// TIA Portal V21 export
DATA_BLOCK "Trend"   // DB5
{ S7_Optimized_Access := 'TRUE' }
// stored: MemoryReserve 100
   VAR
      T : Array[0.."K_NumTrends"] of "Std_Trend";
   END_VAR
BEGIN
   T[0].Valore1 := 0.0;
   T[0].Valore2 := 0.0;
   T[0].Valore3 := 0.0;
   T[0].Valore4 := 0.0;
   T[0].Valore5 := 0.0;
   T[0].Valore6 := 0.0;
   T[0].Valore7 := 0.0;
   T[0].Valore8 := 0.0;
   T[0].AsseY_SinistroMin := 0;
   T[0].AsseY_SinistroMax := 0;
   T[0].AsseY_DestroMin := 0;
   T[0].AsseY_DestroMax := 0;
END_DATA_BLOCK
